TYPE ST_Analog_HWI :
STRUCT
  bTUnderRange      : BOOL;
  bTOverRange       : BOOL;
  bTLimit1          : BOOL;
  bTLimit2          : BOOL;
  bTError           : BOOL;
  siAnaRaw          : INT;  
END_STRUCT
END_TYPE

(* stored: Version 1.1.0.1, ProductVersion 3.1.4024.12
   DUT ST_Analog_HWI: Id {dab81212-4fc8-4bfa-ad28-4b5e5a7bc20f} *)
